// TIA Portal V20 export
TYPE "LER_typeTwoWayActCommand"
// stored: Access Published
   STRUCT
      home : Bool;
      work : Bool;
   END_STRUCT;
END_TYPE
